INTERFACE I_Cylinder

PROPERTY bIsExtend : BOOL
GET
END_GET
END_PROPERTY

PROPERTY bIsRetract : BOOL
GET
END_GET
END_PROPERTY

METHOD Extend : BOOL
VAR_INPUT
END_VAR
END_METHOD

METHOD Retract : BOOL
VAR_INPUT
END_VAR
END_METHOD

END_INTERFACE

(* stored: Version 1.1.0.1, ProductVersion 3.1.4024.12
   Itf I_Cylinder: Id {90982fa2-f182-413f-9fb2-d8a232658566}
   Property bIsExtend: Id {445c20e1-d570-4dff-8efb-092a311630cf}
   Get Get: Id {ac59b736-eec7-4995-83ab-92fd7b15943f}
   Property bIsRetract: Id {d125ba91-5851-4c2d-8123-35bcb38f17f8}
   Get Get: Id {16f5ebf5-44de-4b2d-89b7-1161bb94e694}
   Method Extend: Id {91d98c47-3d9a-4bb9-a3a8-1accebb95519}
   Method Retract: Id {a4852e2c-c128-47c2-8324-e45b99ad198f} *)
